(* PLC project Beremiz non-standard POUs library, Beremiz Beremiz 0.0 *)
(* stored: creationDateTime 2008-12-14T16:53:26, modificationDateTime 2022-12-16T11:59:30 *)

FUNCTION_BLOCK python_eval
  VAR_INPUT
    TRIG : BOOL;
    CODE : STRING;
  END_VAR
  VAR_OUTPUT
    ACK : BOOL;
    RESULT : STRING;
  END_VAR
  VAR
    STATE : DWORD;
    BUFFER : STRING;
    PREBUFFER : STRING;
    TRIGM1 : BOOL;
    TRIGGED : BOOL;
  END_VAR

            {extern void __PythonEvalFB(int, PYTHON_EVAL*);__PythonEvalFB(0, data__);}
          
END_FUNCTION_BLOCK

FUNCTION_BLOCK csv_read_by_string
  VAR_EXTERNAL
    pyext_csv_update : BOOL;
  END_VAR
  VAR_OUTPUT
    ACK : BOOL;
    RESULT : STRING;
  END_VAR
  VAR_INPUT
    FILE_NAME : STRING;
    ROW : STRING;
    COLUMN : STRING;
  END_VAR
  VAR
    OLDCODE : STRING;
    py_eval : python_eval;
    R_TRIG0 : R_TRIG;
    R_TRIG1 : R_TRIG;
    SR0 : SR;
  END_VAR
  VAR  (* added by the conversion: wires and edge detectors of the diagram *)
    _OR15_OUT : BOOL;
    R_TRIG1_2 : R_TRIG;
  END_VAR

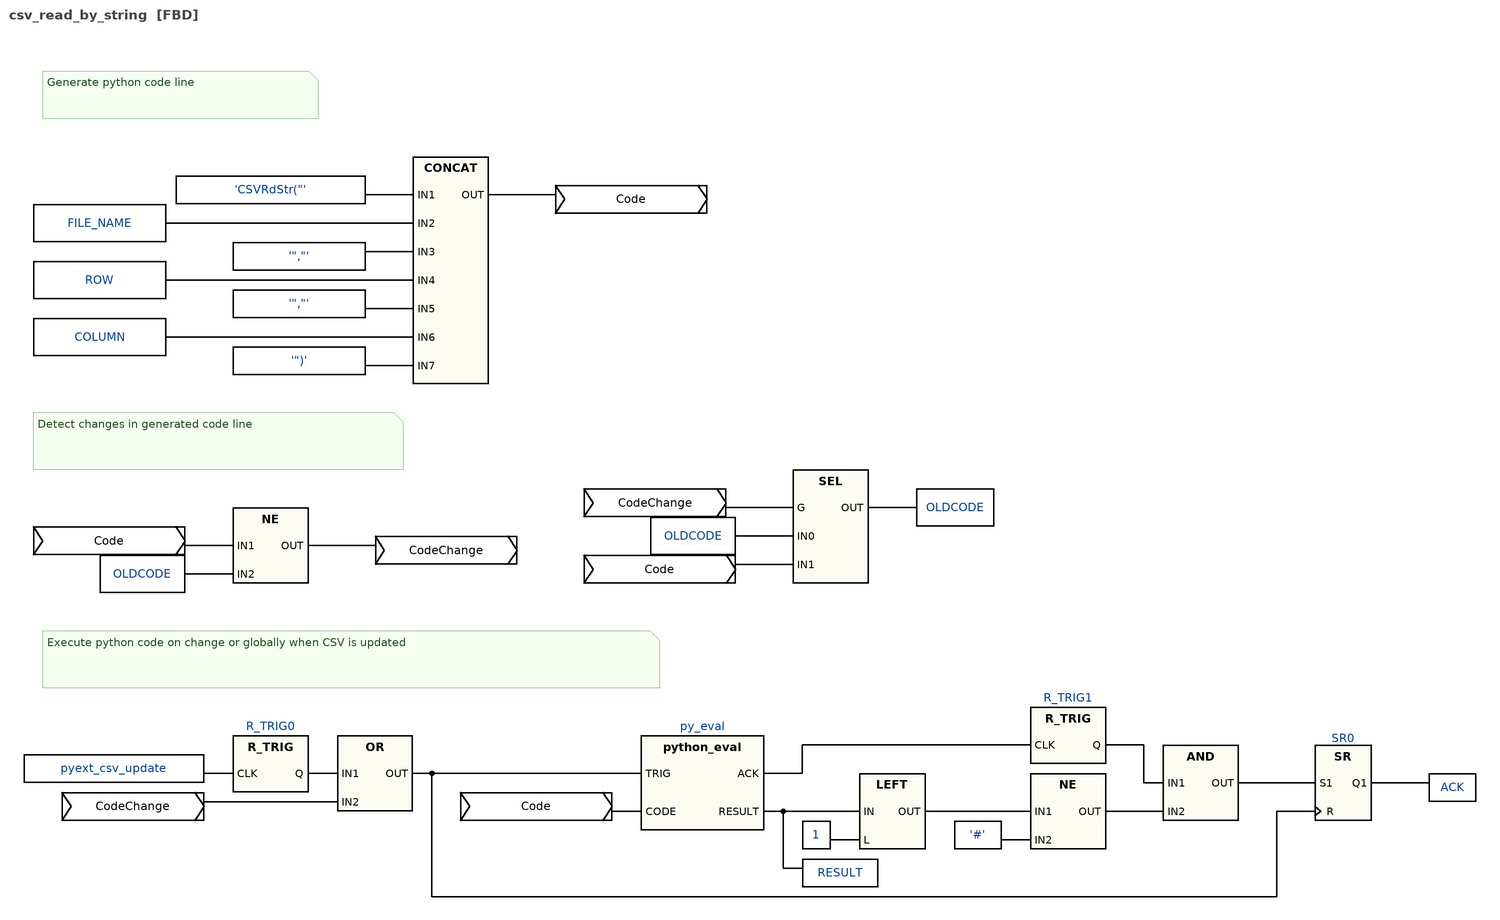
(* FBD diagram, written out as Structured Text *)
(* Generate python code line *)
(* Detect changes in generated code line *)
OLDCODE := SEL(CONCAT('CSVRdStr("', FILE_NAME, '","', ROW, '","', COLUMN, '")') <> OLDCODE, OLDCODE, CONCAT('CSVRdStr("', FILE_NAME, '","', ROW, '","', COLUMN, '")'));
(* Execute python code on change or globally when CSV is updated *)
R_TRIG0(CLK := pyext_csv_update);
_OR15_OUT := R_TRIG0.Q OR CONCAT('CSVRdStr("', FILE_NAME, '","', ROW, '","', COLUMN, '")') <> OLDCODE;
py_eval(TRIG := _OR15_OUT, CODE := CONCAT('CSVRdStr("', FILE_NAME, '","', ROW, '","', COLUMN, '")'));
R_TRIG1(CLK := py_eval.ACK);
R_TRIG1_2(CLK := _OR15_OUT);
SR0(S1 := R_TRIG1.Q AND LEFT(py_eval.RESULT, 1) <> '#', R := R_TRIG1_2.Q);
ACK := SR0.Q1;
RESULT := py_eval.RESULT;
END_FUNCTION_BLOCK

FUNCTION_BLOCK csv_reload
  VAR_EXTERNAL
    pyext_csv_update : BOOL;
  END_VAR
  VAR_OUTPUT
    ACK : BOOL;
    RESULT : STRING;
  END_VAR
  VAR
    py_eval : python_eval;
  END_VAR
  VAR_INPUT
    TRIG : BOOL;
  END_VAR
  VAR
    R_TRIG0 : R_TRIG;
    F_TRIG0 : F_TRIG;
  END_VAR

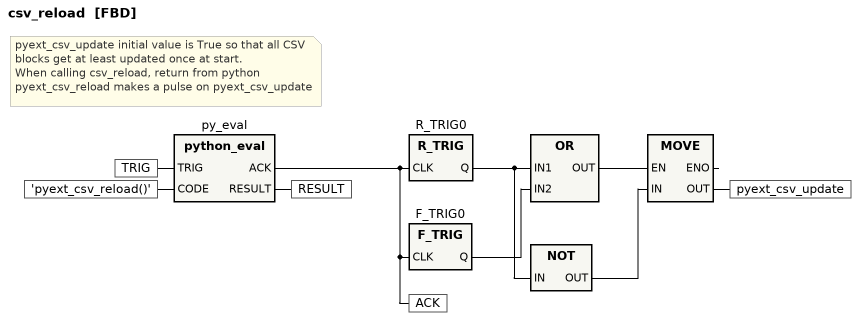
(* FBD diagram, written out as Structured Text *)
(* pyext_csv_update initial value is True so that all CSV blocks get at least updated once at start. 
When calling csv_reload, return from python pyext_csv_reload makes a pulse on pyext_csv_update *)
py_eval(TRIG := TRIG, CODE := 'pyext_csv_reload()');
R_TRIG0(CLK := py_eval.ACK);
F_TRIG0(CLK := py_eval.ACK);
IF R_TRIG0.Q OR F_TRIG0.Q THEN pyext_csv_update := NOT R_TRIG0.Q; END_IF;
ACK := py_eval.ACK;
RESULT := py_eval.RESULT;
END_FUNCTION_BLOCK

FUNCTION_BLOCK csv_read_by_int
  VAR_EXTERNAL
    pyext_csv_update : BOOL;
  END_VAR
  VAR_OUTPUT
    ACK : BOOL;
    RESULT : STRING;
  END_VAR
  VAR_INPUT
    FILE_NAME : STRING;
    ROW : INT;
    COLUMN : INT;
  END_VAR
  VAR
    OLDCODE : STRING;
    py_eval0 : python_eval;
    R_TRIG1 : R_TRIG;
    R_TRIG2 : R_TRIG;
    SR0 : SR;
  END_VAR
  VAR  (* added by the conversion: wires and edge detectors of the diagram *)
    _OR15_OUT : BOOL;
    R_TRIG1_2 : R_TRIG;
  END_VAR

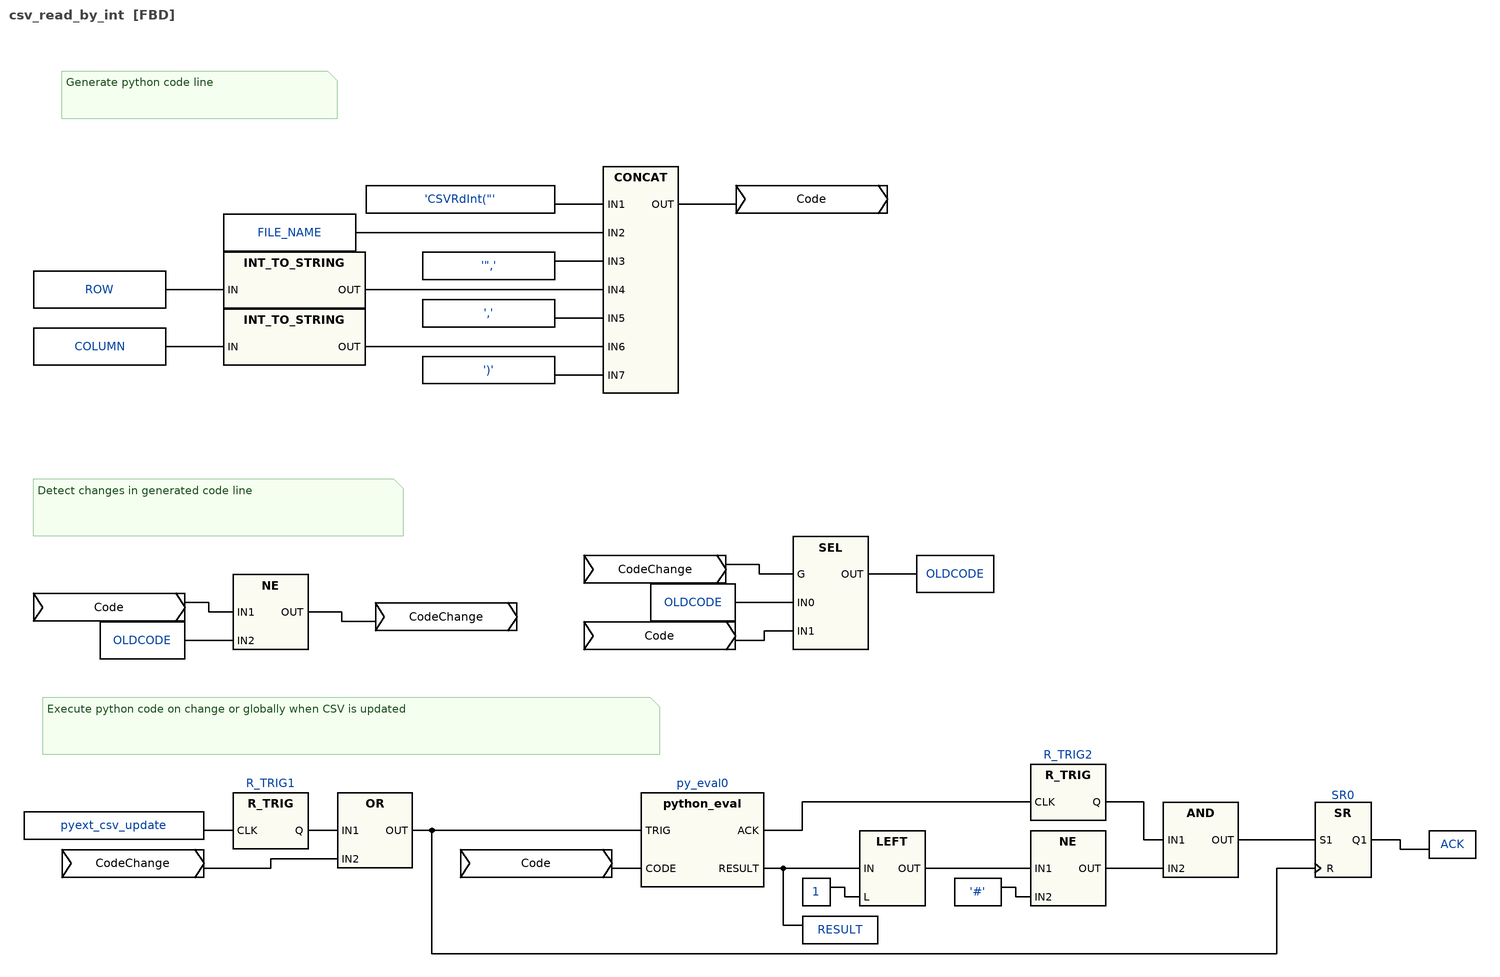
(* FBD diagram, written out as Structured Text *)
(* Generate python code line *)
(* Detect changes in generated code line *)
OLDCODE := SEL(CONCAT('CSVRdInt("', FILE_NAME, '",', INT_TO_STRING(ROW), ',', INT_TO_STRING(COLUMN), ')') <> OLDCODE, OLDCODE, CONCAT('CSVRdInt("', FILE_NAME, '",', INT_TO_STRING(ROW), ',', INT_TO_STRING(COLUMN), ')'));
(* Execute python code on change or globally when CSV is updated *)
R_TRIG1(CLK := pyext_csv_update);
_OR15_OUT := R_TRIG1.Q OR CONCAT('CSVRdInt("', FILE_NAME, '",', INT_TO_STRING(ROW), ',', INT_TO_STRING(COLUMN), ')') <> OLDCODE;
py_eval0(TRIG := _OR15_OUT, CODE := CONCAT('CSVRdInt("', FILE_NAME, '",', INT_TO_STRING(ROW), ',', INT_TO_STRING(COLUMN), ')'));
R_TRIG2(CLK := py_eval0.ACK);
R_TRIG1_2(CLK := _OR15_OUT);
SR0(S1 := R_TRIG2.Q AND LEFT(py_eval0.RESULT, 1) <> '#', R := R_TRIG1_2.Q);
ACK := SR0.Q1;
RESULT := py_eval0.RESULT;
END_FUNCTION_BLOCK

FUNCTION_BLOCK python_poll
  VAR_INPUT
    TRIG : BOOL;
    CODE : STRING;
  END_VAR
  VAR_OUTPUT
    ACK : BOOL;
    RESULT : STRING;
  END_VAR
  VAR
    STATE : DWORD;
    BUFFER : STRING;
    PREBUFFER : STRING;
    TRIGM1 : BOOL;
    TRIGGED : BOOL;
  END_VAR

            {extern void __PythonEvalFB(int, PYTHON_EVAL*);__PythonEvalFB(1,(PYTHON_EVAL*)(void*)data__);}
          
END_FUNCTION_BLOCK

FUNCTION_BLOCK python_gear
  VAR_INPUT
    N : UINT;
    TRIG : BOOL;
    CODE : STRING;
  END_VAR
  VAR_OUTPUT
    ACK : BOOL;
    RESULT : STRING;
  END_VAR
  VAR
    py_eval : python_eval;
    COUNTER : UINT;
  END_VAR
  VAR  (* added by the conversion: wires and edge detectors of the diagram *)
    _ADD10_OUT : UINT;
    _EQ13_OUT : BOOL;
  END_VAR

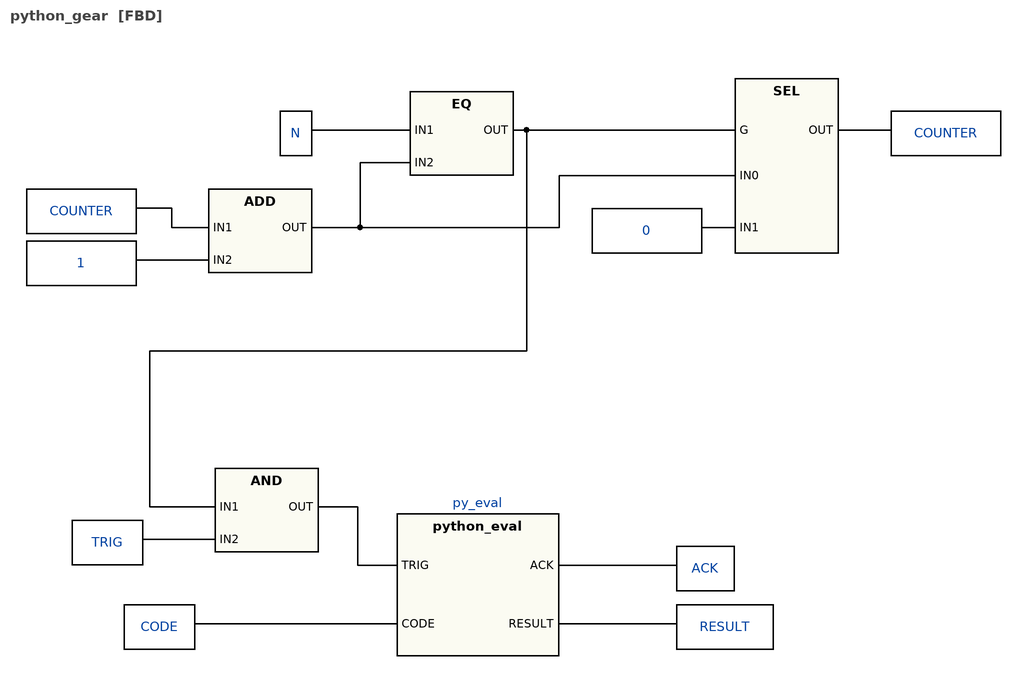
(* FBD diagram, written out as Structured Text *)
_ADD10_OUT := COUNTER + 1;
_EQ13_OUT := N = _ADD10_OUT;
COUNTER := SEL(_EQ13_OUT, _ADD10_OUT, 0);
py_eval(TRIG := _EQ13_OUT AND TRIG, CODE := CODE);
ACK := py_eval.ACK;
RESULT := py_eval.RESULT;
END_FUNCTION_BLOCK

CONFIGURATION configuration0
  VAR_GLOBAL
    pyext_csv_update : BOOL := TRUE;
  END_VAR
END_CONFIGURATION
